// TIA Portal project "w1_BT2" (V14)

(* hardware
DEVICE "S7-1200 station_1"  S7-1200 Station
   slot 0: "Rack_0"  S7-1200 Rack  Rack  V1.0
   slot 1: "PLC_1"  CPU 1214C DC/DC/DC  6ES7 214-1AG40-0XB0  V4.2
*)

// ===== PLC "PLC_1"  CPU 1214C DC/DC/DC =====

VAR_GLOBAL   // PLC tag table "Default tag table"
   "Tag_1" AT %Q0.0 : Bool;
   "Tag_2" AT %Q0.1 : Bool;
   "Tag_3" AT %Q0.2 : Bool;
   "Tag_4" AT %I0.0 : Bool;
   "Tag_5" AT %I0.1 : Bool;
   "Tag_6" AT %I0.2 : Bool;
   "Tag_7" AT %I0.3 : Bool;
   "Tag_8" AT %M0.0 : Bool;
   "Tag_9" AT %I0.4 : Bool;
END_VAR

ORGANIZATION_BLOCK "Main"   // OB1, LAD, ProgramCycle
TITLE = "Main Program Sweep (Cycle)"
{ S7_Optimized_Access := 'TRUE' }
VERSION : 0.1
   VAR_INPUT
      Initial_Call : Bool;   // Initial call of this OB
      Remanence : Bool;   // =True, if remanent data are available
   END_VAR
BEGIN

REGION Network 1
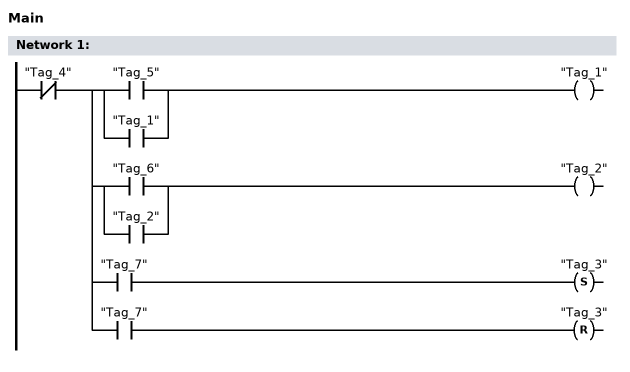
   RUNG wire#powerrail
      I_Contact( "Tag_4" )
      wire#w1
      Contact( "Tag_5" )
      wire#w2
      Coil( "Tag_1" )
   END_RUNG
   RUNG wire#w1
      Contact( "Tag_1" )
   END_RUNG wire#w2
   RUNG wire#w1
      Contact( "Tag_6" )
      wire#w3
      Coil( "Tag_2" )
   END_RUNG
   RUNG wire#w1
      Contact( "Tag_2" )
   END_RUNG wire#w3
   RUNG wire#w1
      Contact( "Tag_7" )
      S_Coil( "Tag_3" )
   END_RUNG
   RUNG wire#w1
      Contact( "Tag_7" )
      R_Coil( "Tag_3" )
   END_RUNG
   // the same network as SCL:
   "Tag_1" := NOT "Tag_4" AND ("Tag_5" OR "Tag_1");
   "Tag_2" := NOT "Tag_4" AND ("Tag_6" OR "Tag_2");
   IF NOT "Tag_4" AND "Tag_7" THEN
       "Tag_3" := TRUE;
       "Tag_3" := FALSE;
   END_IF;
END_REGION
END_ORGANIZATION_BLOCK